PROGRAM MAIN
VAR
	client : HttpClient;
END_VAR

client();

END_PROGRAM

(* stored: Version 1.1.0.1, ProductVersion 3.1.4022.12
   POU MAIN: Id {7d444f4f-0d00-411e-888e-132e3af9a8ac}, SpecialFunc None *)
